FUNCTION_BLOCK ControllerFB (* Template for an empty basic function block *)
  (* Standard: 61499-2 *)
  (* Version 1.0, 2019-03-19, Duc Do Tran, OFFIS e.V. *)
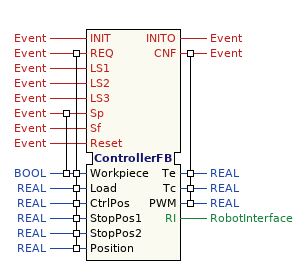
  EVENT_INPUT
    INIT;
    REQ WITH StopPos1, Position, CtrlPos, StopPos2, Load, Workpiece;
    LS1;
    LS2;
    LS3;
    Sp WITH Workpiece;
    Sf;
    Reset;
  END_EVENT
  EVENT_OUTPUT
    INITO;
    CNF WITH Te, Tc, PWM;
  END_EVENT
  VAR_INPUT
    Workpiece : BOOL;
    Load : REAL;
    CtrlPos : REAL := 15;
    StopPos1 : REAL := 90;
    StopPos2 : REAL := 180;
    Position : REAL;
  END_VAR
  VAR_OUTPUT
    Te : REAL;
    Tc : REAL;
    PWM : REAL;
  END_VAR
  PLUGS
    RI : RobotInterface;
  END_PLUGS
  VAR
    t0 : TIME; (* Internal Variable *)
    bd : BOOL; (* Internal Variable *)
    flag : BOOL; (* Internal Variable *)
    t : REAL; (* Internal Variable *)
    unique : BOOL := TRUE; (* Internal Variable *)
    i : USINT; (* Internal Variable *)
    Pos0 : REAL; (* Internal Variable *)
    LimPos : REAL; (* Internal Variable *)
    DirRot : BOOL; (* Internal Variable *)
  END_VAR
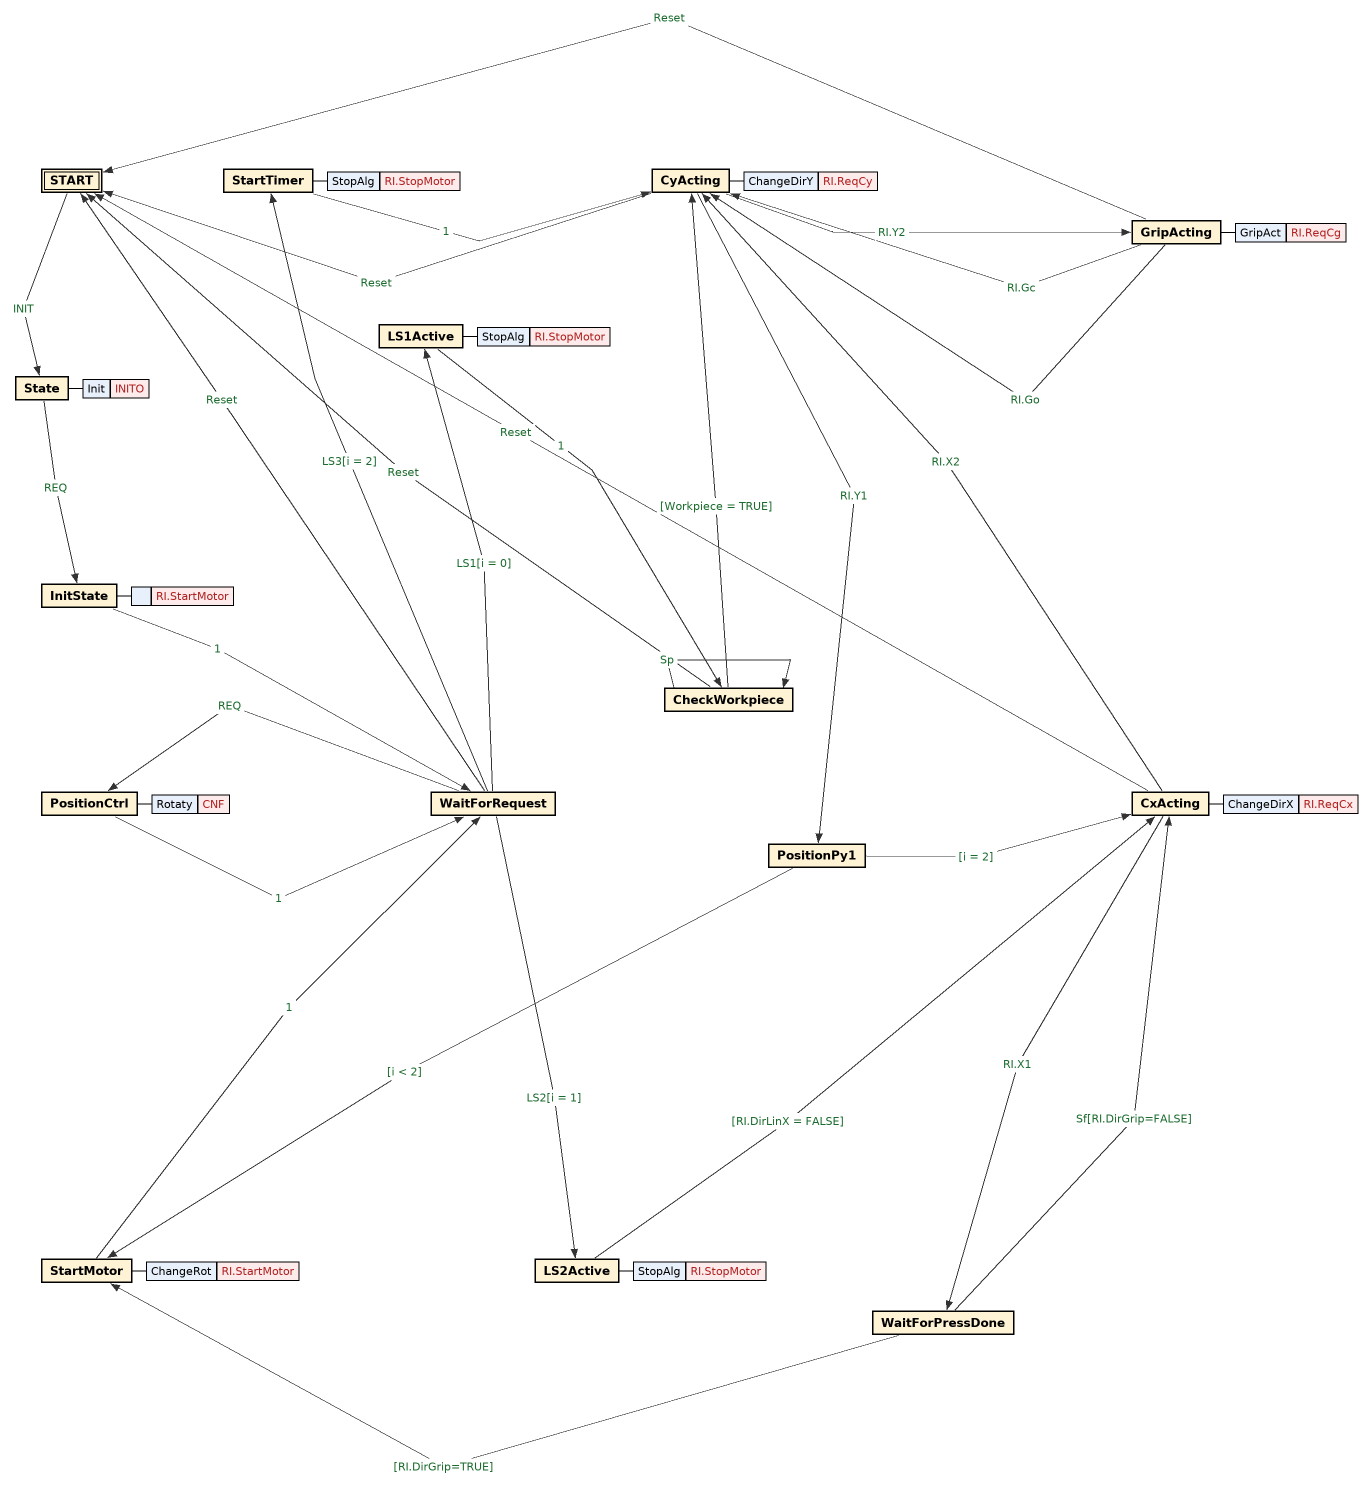
  EC_STATES
    START; (* Initial State *)
    StartTimer : StopAlg -> RI.StopMotor;
    GripActing : GripAct -> RI.ReqCg;
    WaitForPressDone;
    LS1Active : StopAlg -> RI.StopMotor;
    InitState : -> RI.StartMotor;
    WaitForRequest;
    PositionCtrl : Rotaty -> CNF;
    LS2Active : StopAlg -> RI.StopMotor;
    CyActing : ChangeDirY -> RI.ReqCy;
    CxActing : ChangeDirX -> RI.ReqCx;
    PositionPy1;
    CheckWorkpiece;
    StartMotor : ChangeRot -> RI.StartMotor;
    State : Init -> INITO;
  END_STATES
  EC_TRANSITIONS
    InitState TO WaitForRequest := 1;
    PositionCtrl TO WaitForRequest := 1;
    WaitForRequest TO LS1Active := LS1[i = 0];
    WaitForRequest TO LS2Active := LS2[i = 1];
    CyActing TO GripActing := RI.Y2;
    GripActing TO CyActing := RI.Gc;
    LS2Active TO CxActing := [RI.DirLinX = FALSE];
    CxActing TO CyActing := RI.X2;
    GripActing TO CyActing := RI.Go;
    CxActing TO WaitForPressDone := RI.X1;
    WaitForRequest TO StartTimer := LS3[i = 2];
    WaitForRequest TO PositionCtrl := REQ;
    StartTimer TO CyActing := 1;
    CyActing TO PositionPy1 := RI.Y1;
    PositionPy1 TO CxActing := [i = 2];
    WaitForPressDone TO CxActing := Sf[RI.DirGrip=FALSE];
    CheckWorkpiece TO CyActing := [Workpiece = TRUE];
    CheckWorkpiece TO CheckWorkpiece := Sp;
    LS1Active TO CheckWorkpiece := 1;
    WaitForPressDone TO StartMotor := [RI.DirGrip=TRUE];
    PositionPy1 TO StartMotor := [i < 2];
    StartMotor TO WaitForRequest := 1;
    WaitForRequest TO START := Reset;
    CyActing TO START := Reset;
    CxActing TO START := Reset;
    GripActing TO START := Reset;
    State TO InitState := REQ;
    START TO State := INIT;
    CheckWorkpiece TO START := Reset;
  END_TRANSITIONS
  ALGORITHM GripAct IN ST: (* new algorithm *)
//Load := LoadIn;
RI.DirGrip := NOT (RI.DirGrip);
IF (RI.DirGrip = TRUE) THEN
	RI.LoadIn := Load;
ELSE
	RI.LoadIn := 0;
END_IF;
  END_ALGORITHM
  ALGORITHM Rotaty IN ST: (* new algorithm *)
IF (unique = TRUE) THEN
	unique := FALSE;
	IF (Position >= StopPos2 ) THEN
			DirRot := FALSE;
	END_IF;
END_IF;
IF(bd = TRUE) THEN
	t0 := NOW_MONOTONIC();
	flag := FALSE;
	bd := FALSE;
END_IF;
IF (DirRot = FALSE) THEN
	IF (Position <= LimPos - CtrlPos) THEN
		PWM := 1;
	ELSE
		PWM := 0.5;
		IF (flag = FALSE) THEN
			flag := TRUE;
			t := TIME_IN_S_TO_LREAL(NOW_MONOTONIC()- t0);
		END_IF;
	END_IF;
ELSE
	IF ( Position >= LimPos + CtrlPos) THEN
		PWM := -1;
	ELSE
		PWM := -0.5;
		IF (flag = FALSE) THEN
			flag := TRUE;
			t := TIME_IN_S_TO_LREAL(NOW_MONOTONIC()- t0);
		END_IF;
	END_IF;
END_IF;
Tc := t;
  END_ALGORITHM
  ALGORITHM Init IN ST: (* new algorithm *)
bd := TRUE;
DirRot := TRUE;
RI.DirLinX := FALSE;
RI.DirLinY := FALSE;
RI.DirGrip := FALSE;
LimPos := 0;
i := 0;
  END_ALGORITHM
  ALGORITHM StopAlg IN ST: (* new algorithm *)
PWM := 0;
i :=( i + 1) MOD 3;
Te := TIME_IN_S_TO_LREAL(NOW_MONOTONIC()- t0);
  END_ALGORITHM
  ALGORITHM ChangeDirX IN ST: (* new algorithm *)
RI.DirLinX := NOT(RI.DirLinX);
  END_ALGORITHM
  ALGORITHM ChangeDirY IN ST: (* new algorithm *)
RI.DirLinY := NOT(RI.DirLinY);
  END_ALGORITHM
  ALGORITHM ChangeRot IN ST: (* new algorithm *)
IF (i = 0) THEN
	DirRot := TRUE;
	LimPos := 0;
ELSE
	DirRot := FALSE;
	IF (i = 1) THEN
		LimPos := StopPos1;
	ELSE
		LimPos := StopPos2;
	END_IF;
END_IF;
bd := TRUE;
flag := FALSE;
  END_ALGORITHM
END_FUNCTION_BLOCK
